(* Logix 5000 project; controller EuniceF_ICA11 vendor 1 type 14 code 150 rev 37.11; software revision 37.00 *)

TASK MainTask (continuous, watchdog 500 ms) : MainProgram

MODULES
   Local : vendor 1 type 14 code 150 (Compact 0, rev 37.11)
      Discrete_IO : Embedded (Compact 1, rev 3.1, Output RPI 20 ms)
      Analog_IO : Embedded (Compact 2, rev 1.1, Output RPI 80 ms)
      Counters : Embedded (Compact 3, rev 1.1, Output RPI 20 ms)
END_MODULES

VAR_GLOBAL   (* controller tags *)
   ALERT1 : ALIAS FOR Local:1:O.Data.2;
   CAMERA : ALIAS FOR Local:1:I.Data.15;
   E_RUN : ALIAS FOR Local:1:O.Data.1;
   ESCALATOR : ALIAS FOR Local:1:O.Data.1;
   L_STOP : ALIAS FOR Local:1:I.Data.10;
   START : ALIAS FOR Local:1:I.Data.11;
   STOP : ALIAS FOR Local:1:I.Data.8;
   TIMER1 : TIMER := (PRE := 3000);
   U_STOP : ALIAS FOR Local:1:I.Data.9;
END_VAR

PROGRAM MainProgram   (* main routine MainRoutine *)
VAR
   ALERT : BOOL;
END_VAR

ROUTINE MainRoutine   (* ladder *)
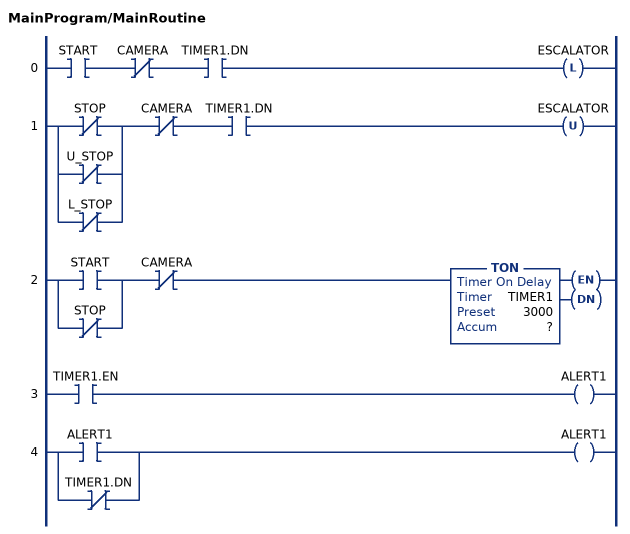
   0: XIC(START)XIO(CAMERA)XIC(TIMER1.DN)OTL(ESCALATOR);
   1: [XIO(STOP) ,[XIO(U_STOP) ,XIO(L_STOP) ] ]XIO(CAMERA)XIC(TIMER1.DN)OTU(ESCALATOR);
   2: [XIC(START) ,XIO(STOP) ]XIO(CAMERA)TON(TIMER1,?,?);
   3: XIC(TIMER1.EN)OTE(ALERT1);
   4: [XIC(ALERT1) ,XIO(TIMER1.DN) ]OTE(ALERT1);
END_ROUTINE
END_PROGRAM
